TYPE Vec3i : ARRAY[1..3] OF INT; END_TYPE

(* stored: Version 1.1.0.1, ProductVersion 3.1.4024.11
   DUT Vec3i: Id {316d763a-61a9-414f-804f-221cc8dd7193} *)
